(* IEC 61131-3 sources: repolevel_ST_code_completion/real_groud_truth最新/repoeval_ProductionLine/readful_result, 6 files *)

(* ---- Motor.st ---- *)
VAR
	WaitTimer:TON;
	InternalSequenceDelay:TIME;
END_VAR

METHOD TurnOn : BOOL
VAR_INPUT
	MotorI:MotorI;
END_VAR
VAR_OUTPUT
	MotorO:MotorO;
END_VAR
VAR
	WaitTimer:TON;
	InternalSequenceDelay:TIME;
END_VAR

IF MotorO.FaultStatus = FALSE THEN
	WaitTimer(IN:=TRUE, PT:=InternalSequenceDelay);
END_IF

IF WaitTimer.Q THEN
	MotorO.Coil := TRUE;
	WaitTimer(IN := FALSE);
END_IF

METHOD TurnOff : BOOL
VAR_INPUT
	MotorI:MotorI;
END_VAR
VAR_OUTPUT
	MotorO:MotorO;
END_VAR
VAR
	WaitTimer:TON;
	InternalSequenceDelay:TIME;
END_VAR

MotorO.Coil := FALSE;

METHOD SetFault : BOOL
VAR_INPUT
	MotorI:MotorI;
END_VAR
VAR_OUTPUT
	MotorO:MotorO;
END_VAR
VAR
	WaitTimer:TON;
	InternalSequenceDelay:TIME;
END_VAR

IF MotorI.Overload THEN
	MotorO.FaultStatus := TRUE;
	TurnOff();
END_IF

METHOD SetWaitTime : BOOL
VAR_INPUT
	MotorI:MotorI;
	SequenceDelay:TIME;
END_VAR
VAR_OUTPUT
	MotorO:MotorO;
END_VAR
VAR
	WaitTimer:TON;
	InternalSequenceDelay:TIME;
END_VAR

InternalSequenceDelay := SequenceDelay;

PROGRAM PLC_PRG
VAR
	Motor:Motor;
	MotorInputs:MotorI;
	MotorOutputs:MotorO;
	liga: BOOL;
	desliga: BOOL;
	settime: BOOL;
	setfault: BOOL;
	reset: BOOL;
	timetemp: TIME;
END_VAR

Motor(MotorI := MotorInputs, MotorO => MotorOutputs);

IF liga THEN
	Motor.TurnOn();
	liga := FALSE;
END_IF

IF desliga THEN
	Motor.TurnOff();
	desliga := FALSE;
END_IF

IF settime THEN
	Motor.SetWaitTime(SequenceDelay := timetemp);
	settime := FALSE;
END_IF

IF setfault THEN
	Motor.SetFault();
	setfault := FALSE;
END_IF

IF reset THEN
	MotorO.FaultStatus := FALSE;
	reset := FALSE;
END_IF

(* ---- Motor_ResetFault.st ---- *)
VAR
	WaitTimer:TON;
	InternalSequenceDelay:TIME;
	ResetDetect:R_TRIG;
END_VAR

// Detect the rising edge of the FaultReset signal
ResetDetect(CLK := MotorI.FaultReset);

// If a reset is detected, clear the fault status
IF ResetDetect.Q THEN
	MotorO.FaultStatus := FALSE;
END_IF;

// Return TRUE to indicate the method executed successfully
ResetFault := TRUE;

(* ---- Motor_SetFault.st ---- *)
VAR
	WaitTimer:TON;
	InternalSequenceDelay:time;
END_VAR

IF MotorI.Overload THEN
	MotorO.FaultStatus := TRUE;
	TurnOff();
END_IF

(* ---- Motor_SetWaitTime.st ---- *)
VAR
	WaitTimer:TON;
	InternalSequenceDelay:TIME;
END_VAR

// Assign the input SequenceDelay to the internal variable
InternalSequenceDelay := SequenceDelay;

// Check if the motor is not in a fault state before setting the wait time
IF MotorO.FaultStatus = FALSE THEN
	// Configure the timer with the provided delay
	WaitTimer(IN := TRUE, PT := InternalSequenceDelay);

	// If the timer has elapsed, reset the timer and return TRUE
	IF WaitTimer.Q THEN
		WaitTimer(IN := FALSE);
		RETURN TRUE;
	END_IF;
ELSE
	// If the motor is in a fault state, do not set the wait time
	RETURN FALSE;
END_IF;

(* ---- Motor_TurnOff.st ---- *)
VAR
	WaitTimer:TON;
	InternalSequenceDelay:time;
END_VAR

MotorO.Coil := FALSE;
RETURN TRUE;

(* ---- Motor_TurnOn.st ---- *)
VAR
	WaitTimer:TON;
	InternalSequenceDelay:time;
END_VAR

// Check if the motor is not in a fault state
IF MotorO.FaultStatus = FALSE THEN
	// Start the timer for the internal sequence delay
	WaitTimer(IN:=TRUE, PT:=InternalSequenceDelay);
END_IF

// If the timer has elapsed, turn on the motor coil
IF WaitTimer.Q THEN
	MotorO.Coil := TRUE;
	// Stop the timer
	WaitTimer(IN:=FALSE);
END_IF

// Return the status of the motor coil as the method's result
RETURN MotorO.Coil;
